ABB RAPID module: MainModule.mod

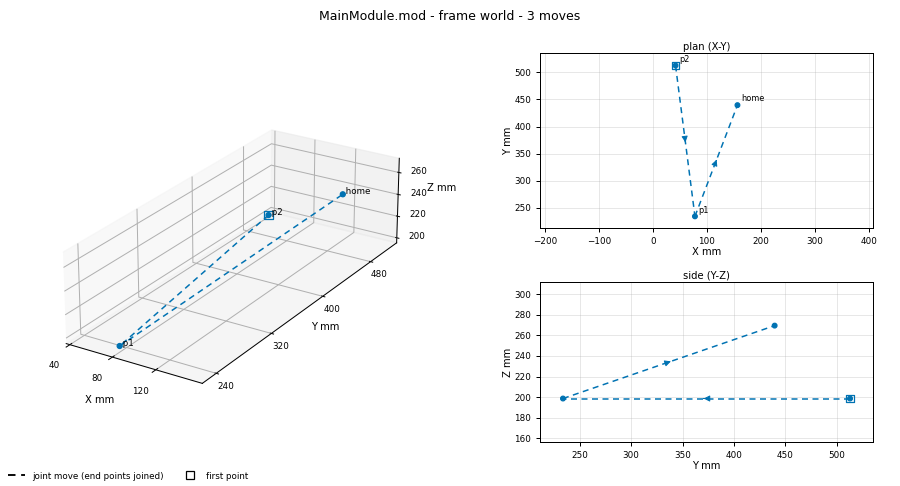
[picture p0: tool path of MainModule.mod in frame world, 3 of 3 moves have a stored position in this frame; points joined in program order, loops and branches not executed]
MODULE MainModule
	CONST robtarget home:=[[156.39,439.53,269.48],[0.0660091,0.84242,-0.111214,0.523071],[0,0,-1,4],[103.219,9E+9,9E+9,9E+9,9E+9,9E+9]];
	CONST robtarget p1:=[[77.76,233.84,198.63],[0.0660096,0.84242,-0.111214,0.523071],[0,0,0,4],[101.964,9E+9,9E+9,9E+9,9E+9,9E+9]];
	CONST robtarget p2:=[[41.88,512.79,198.63],[0.0660095,0.84242,-0.111214,0.523071],[0,0,0,4],[101.964,9E+9,9E+9,9E+9,9E+9,9E+9]];
	PROC main()
		MoveJ p2, v1000, z50, tool0;
		MoveJ p1, v1000, z50, tool0;
		MoveJ home, v1000, z50, tool0;
	ENDPROC
ENDMODULE
